// TIA Portal V17 export
// export: Created 2026-05-13T16:29:31.5238933Z, ExportSetting WithDefaults, DisplayName Totally Integrated Automation Portal, DisplayVersion V17 Update 4, DisplayName TIA Portal Openness, DisplayVersion V17 Update 4, DisplayName TIA Portal Version Control Interface, DisplayVersion V17, DisplayName SINAMICS Startdrive Advanced, DisplayVersion V17, DisplayName SINAMICS Startdrive G130, G150, S120, S150, SINAMICS MV, S210, DisplayVersion V17, DisplayName SINAMICS Startdrive G110M, G120, G120C, G120D, G120P, G115D, DisplayVersion V17, DisplayName STEP 7 Professional, DisplayVersion V17 Update 4, DisplayName STEP 7 Safety, DisplayVersion V17, DisplayName WinCC Professional, DisplayVersion V17 Update 4
TagTable "Codex_Popup_PLC_Named_Int_Tags"
  DB_Components_Valve01_ClickTrig : Int  (1 s, start 0)   // Maps to DB_Components.Valve01.ClickTrig.
  DB_Components_Valve01_DoubleClickTime : Int  (1 s, start 800)   // Maps to DB_Components.Valve01.DoubleClickTime.
  DB_Components_Valve01_Switch1 : Int  (1 s, start 0)   // Maps to DB_Components.Valve01.Switch[1].
  DB_Components_Valve01_RealValue1_Int : Int  (1 s, start 0)   // Integer placeholder for DB_Components.Valve01.RealValue[1].
  DB_ActivePopup_Valve01_Visible : Bool  (PLC tag DB_ActivePopup.Valve01.Visible, HMI_连接_1, 1 s, start 0)   // Maps to DB_ActivePopup.Valve01.Visible.
  DB_ActivePopup_Valve01_ActiveID : Int  (1 s, start 1)   // Maps to DB_ActivePopup.Valve01.ActiveID.
  DB_ActivePopup_Valve01_Confirmed : Bool  (PLC tag DB_ActivePopup.Valve01.Confirmed, HMI_连接_1, 1 s, start 0)   // Maps to DB_ActivePopup.Valve01.Confirmed.
  DB_ActivePopup_Valve01_ConfirmBtn : Int  (1 s, start 0)   // Maps to DB_ActivePopup.Valve01.ConfirmBtn.
  DB_ActivePopup_Valve01_CancelBtn : Int  (1 s, start 0)   // Maps to DB_ActivePopup.Valve01.CancelBtn.
  DB_Components_Heater01_ClickTrig : Int  (1 s, start 0)   // Maps to DB_Components.Heater01.ClickTrig.
  DB_Components_Heater01_DoubleClickTime : Int  (1 s, start 800)   // Maps to DB_Components.Heater01.DoubleClickTime.
  DB_Components_Heater01_Switch1 : Int  (1 s, start 0)   // Maps to DB_Components.Heater01.Switch[1].
  DB_Components_Heater01_RealValue1_Int : Int  (1 s, start 0)   // Integer placeholder for DB_Components.Heater01.RealValue[1].
  DB_ActivePopup_Heater01_Visible : Int  (1 s, start 0)   // Maps to DB_ActivePopup.Heater01.Visible.
  DB_ActivePopup_Heater01_Confirmed : Int  (1 s, start 0)   // Maps to DB_ActivePopup.Heater01.Confirmed.
  DB_ActivePopup_Heater01_ConfirmBtn : Int  (1 s, start 0)   // Maps to DB_ActivePopup.Heater01.ConfirmBtn.
  DB_ActivePopup_Heater01_CancelBtn : Int  (1 s, start 0)   // Maps to DB_ActivePopup.Heater01.CancelBtn.
  DB_Components_Fan01_ClickTrig : Int  (1 s, start 0)   // Maps to DB_Components.Fan01.ClickTrig.
  DB_Components_Fan01_DoubleClickTime : Int  (1 s, start 800)   // Maps to DB_Components.Fan01.DoubleClickTime.
  DB_Components_Fan01_Switch1 : Int  (1 s, start 0)   // Maps to DB_Components.Fan01.Switch[1].
  DB_Components_Fan01_RealValue1_Int : Int  (1 s, start 0)   // Integer placeholder for DB_Components.Fan01.RealValue[1].
  DB_ActivePopup_Fan01_Visible : Int  (1 s, start 0)   // Maps to DB_ActivePopup.Fan01.Visible.
  DB_ActivePopup_Fan01_ActiveID : Int  (1 s, start 3)   // Maps to DB_ActivePopup.Fan01.ActiveID.
  DB_ActivePopup_Fan01_Confirmed : Int  (HMI_连接_1, 1 s, start 0)   // Maps to DB_ActivePopup.Fan01.Confirmed.
  DB_ActivePopup_Fan01_ConfirmBtn : Int  (1 s, start 0)   // Maps to DB_ActivePopup.Fan01.ConfirmBtn.
  DB_ActivePopup_Fan01_CancelBtn : Int  (1 s, start 0)   // Maps to DB_ActivePopup.Fan01.CancelBtn.
